// TIA Portal V20 export
TYPE "typeSequenceControlNodeJobInterfaceMonitoring"
// stored: Namespace Unit1.Em3
   STRUCT
      spare { ExternalWritable := 'False'} : Bool;
   END_STRUCT;
END_TYPE
